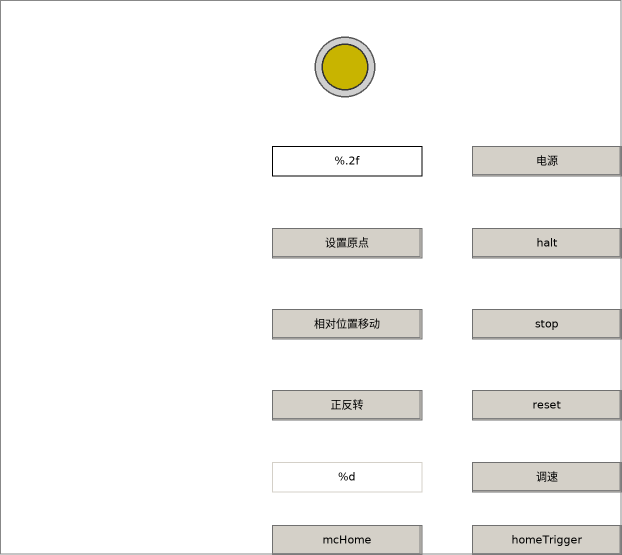
VISUALIZATION singleAxis  // 622x555
    Rectangle (272,146 150x30), "%.2f", text variable: single.axisx.NcToPlc.ActPos
    Button (272,390 150x30), "正反转"
        OnMouseClick: toggle single.jogDirection
        OnMouseClick: execute { single.shouldJog := TRUE; }
    Lamp1 (310,32 70x70), variable: single.axisx.NcToPlc.StateDWord.20, style: Lamp-Lamp1-Yellow
    Button (272,309 150x30), "相对位置移动"
        tap single.shouldMoveRel
    Button (272,228 150x30), "设置原点"
        tap single.shouldSetZero
    Button (472,146 150x30), "电源"
        toggle single.shouldPowerOn
    Button (472,228 150x30), "halt"
        tap single.shouldHalt
    Button (472,309 150x30), "stop"
        tap single.shouldStop
    Button (472,462 150x30), "调速"
        tap single.shouldAdjustVelocity
    Textfield (272,462 150x30), "%d", text variable: single.velocity
        OnMouseClick: write single.velocity via VisuDialogs.Numpad, min 10, max 500
    Button (472,390 150x30), "reset"
        tap single.shouldReset
    Button (272,525 150x30), "mcHome"
        tap single.shouldGoHome
    Button (472,525 150x30), "homeTrigger"
        tap single.homeTrigger
END_VISUALIZATION

(* stored: Version 1.1.0.1, ProductVersion 3.1.4024.4
   Visu singleAxis: Id {be1145ad-d74b-4ba3-bd00-5a0c394b8114} *)
